			IF iRecValveMode <> 63 AND xDownloadDone = FALSE THEN	// The transfer mode is currently not active and the values are not downloaded yet
				// check whether the WebConfig blocks the access to transfer mode
				fbReadBitsFromWord(wData := awBusDataFromVTEM[0], iStartBit := 8, iEndBit := 15, iValue => iAppStatus);
				IF iRecValveMode = 61 AND iAppStatus = 10 THEN 		// access denied by WebConfig
					xDownloadError := TRUE;
					iResponse := eTransferResponse.access_denied_WebConfig;
					iCommandNumber := 3; 			// do nothing (here: command 'stop')
				ELSIF iRecValveMode = 61 AND iAppStatus = 11 THEN 	// access denied due to an active saving process
					xDownloadError := TRUE;
					iResponse := eTransferResponse.access_denied_saving;
					iCommandNumber := 3; 			// do nothing (here: command 'stop')
				ELSIF iRecValveMode = 61 AND iAppStatus = 15 THEN 	// no valve detected
					xDownloadError := TRUE;
					iResponse := eTransferResponse.no_valve_detected; 
					iCommandNumber := 1; 			// keep downloading (here: command 'download') In a Firmware older than 4.16(E) an empty valve keep sending ValveMode 61 and AppStatus 15. In Firmware 4.16(E) the message changes with a tranfer
				ELSIF iRecValveMode = 61 AND iAppStatus = 0 AND xTransferComplete = TRUE THEN
					// All values are downloaded and the transfer mode has been closed properly
					xDownloadDone := TRUE;
					xDownloadError := FALSE;
					iCommandNumber := 3; 			// command 'stop' to remain the valve stopped
				ELSE	// ready to start transfer mode
					xDownloadError := FALSE;
					iResponse := eTransferResponse.transferring;
					iCommandNumber := 1; 			// command 'download' for the current value
				END_IF
		
			ELSIF iRecValveMode = 63 AND xDownloadDone = FALSE THEN		// The transfer mode is active, but the values are not downloaded yet
				fbReadBitsFromWord(wData := awBusDataFromVTEM[0], iStartBit := 8, iEndBit := 12, iValue => iRecChannel);
				fbReadBitsFromWord(wData := awBusDataFromVTEM[0], iStartBit := 13, iEndBit := 15, iValue => iRecTransferCtrl);
				fbReadBitsFromWord(wData := awBusDataFromVTEM[1], iStartBit := 0, iEndBit := 7, iValue => iRecAddressedTargetType);
				fbReadBitsFromWord(wData := awBusDataFromVTEM[1], iStartBit := 8, iEndBit := 15, iValue => iRecIndex);
				iRecTransferValue := WORD_TO_INT(awBusDataFromVTEM[2]);
		 
				IF aTransferPackages[iCurrentValue].iChannel = iRecChannel AND iRecTransferCtrl = 1 AND aTransferPackages[iCurrentValue].iAddressedTarget = iRecAddressedTargetType AND
					aTransferPackages[iCurrentValue].iIndex = iRecIndex AND  aTransferPackages[iCurrentValue].iTransferValue = iRecTransferValue THEN
						// The download command for the parameter was mirrored by the Motion Terminal, the download has been confirmed
						
						xDownloadError := FALSE;
						iCurrentValue := iCurrentValue +1;		// next value
						
						// check whether there is another value
						IF aTransferPackages[iCurrentValue].iAddressedTarget = 0 AND aTransferPackages[iCurrentValue].iChannel = 0 AND aTransferPackages[iCurrentValue].iIndex = 0 AND
							aTransferPackages[iCurrentValue].iTransferValue = 0 THEN 	// last value reached
							
							iCommandNumber := 2; 		// exit transfer mode
							iResponse := eTransferResponse.transfer_successful;
							xTransferComplete := TRUE;
							xStopPending := TRUE;
						ELSE
							iCommandNumber := 1; 		// command 'download' for the (next) value
							iResponse := eTransferResponse.transferring;
						END_IF
					
				ELSIF iRecChannel = 0 AND iRecTransferCtrl = 0 AND iRecAddressedTargetType = 0 AND iRecIndex = 0 AND iRecTransferValue <> 0 AND xFirstCycle = FALSE THEN
					// An invalid command was sent when using the transfer mode
					
					iCommandNumber := 1; 			// command 'download' for the current value
					xDownloadError := TRUE; 
					
					CASE iRecTransferValue OF		// indicates the type of the invalid command
						1: 	iResponse := eTransferResponse.invalid_Channel;
						2: 	iResponse := eTransferResponse.invalid_TransferControl;	// this should never happen
						3: 	iResponse := eTransferResponse.invalid_AddressedTarget;
						4: 	iResponse := eTransferResponse.invalid_Index;
						5: 	iResponse := eTransferResponse.invalid_TransferValue;
						6: 	iResponse := eTransferResponse.invalid_combination;
						7:  iResponse := eTransferResponse.access_denied_DataInUse;
						8:	iResponse := eTransferResponse.no_data_empty_slot;
					END_CASE
					
				ELSE	// A different value is treated in transfer mode or the command was mirrored wrong
					// waiting for stop ack
					IF xStopPending = FALSE THEN
						iCommandNumber := 1; 			// command 'download' for the current value
						xDownloadError := FALSE;
						iResponse := eTransferResponse.transferring;
					END_IF
				END_IF
			
			ELSE // xDownloadDone = TRUE
				IF aTransferPackages[iCurrentValue].iChannel = 0 AND aTransferPackages[iCurrentValue].iAddressedTarget = 0 AND  aTransferPackages[iCurrentValue].iIndex = 0 AND  aTransferPackages[iCurrentValue].iTransferValue = 0 THEN
					// The FB is still active although all values are already downloaded
					iResponse := eTransferResponse.transfer_successful;
					xDownloadError := FALSE;
					iCommandNumber := 3; 		// do nothing (here: command 'stop', MAs remain stopped)
				ELSE
					// Another set of values was inserted to the FB without resetting the internal state with a falling edge at xExecute before
					iResponse := eTransferResponse.FB_needs_rising_edge_xExecute;
					xDownloadError := TRUE;
					iCommandNumber := 2; 		// do nothing (here: command 'exit transfer mode')
				END_IF
			END_IF
		END_IF
		
	ELSE // xInputValid = FALSE OR xInputConsistent = FALSE
		xDownloadDone := FALSE;
		xDownloadError := TRUE;
		IF iRecValveMode = 63 THEN
			iCommandNumber := 2; 				// command 'exit transfer mode'
		ELSE
			iCommandNumber := 3;				// command 'stop'
		END_IF
	END_IF
	
	xFirstCycle := FALSE;

ELSIF xExecute = FALSE AND xFirstCycle = FALSE THEN			// falling edge at input xExecute, resetting the function block
	IF iRecValveMode = 63 THEN
		iCommandNumber := 2;								// exit transfer mode
	ELSE
		xFirstCycle := TRUE;
		xDownloadDone := FALSE;
		xDownloadError := FALSE;
		xTransferComplete := FALSE;
		iCurrentValue := 0;
		xStopPending := FALSE;
		iResponse := eTransferResponse.ready_for_new_transfer;
		iCommandNumber := 0; 								// do nothing (idle)
	END_IF
		
ELSIF xExecute = FALSE AND xFirstCycle = TRUE THEN			// idle mode for the function block
	iResponse := eTransferResponse.ready_for_new_transfer;
	iCommandNumber := 0;
END_IF

CASE iCommandNumber OF
	0: // idle

	1: // download the current value, addressed and specified in the array of values
		fbWriteValueToWord(iValue := 63, iStartBit := 0, iEndBit := 5, wDataWord := awBusDataToVTEM[0]); 												// ValveMode = 63
		fbWriteValueToWord(iValue := 0, iStartBit := 6, iEndBit := 7, wDataWord := awBusDataToVTEM[0]); 												// (empty)
		fbWriteValueToWord(iValue := aTransferPackages[iCurrentValue].iChannel, iStartBit := 8, iEndBit := 12, wDataWord := awBusDataToVTEM[0]); 		// Channel
		fbWriteValueToWord(iValue := 1, iStartBit := 13, iEndBit := 15, wDataWord := awBusDataToVTEM[0]); 												// TransferControl = download
		fbWriteValueToWord(iValue := aTransferPackages[iCurrentValue].iAddressedTarget, iStartBit := 0, iEndBit := 7, wDataWord := awBusDataToVTEM[1]); 	// AddressedTarget
		fbWriteValueToWord(iValue := aTransferPackages[iCurrentValue].iIndex, iStartBit := 8, iEndBit := 15, wDataWord := awBusDataToVTEM[1]); 			// Index
		
		awBusDataToVTEM[2] := INT_TO_WORD(aTransferPackages[iCurrentValue].iTransferValue);
	
	2: // exit transfer mode
		fbWriteValueToWord(iValue := 63, iStartBit := 0, iEndBit := 5, wDataWord := awBusDataToVTEM[0]); 												// ValveMode = 63
		fbWriteValueToWord(iValue := 0, iStartBit := 6, iEndBit := 7, wDataWord := awBusDataToVTEM[0]); 												// (empty)
		fbWriteValueToWord(iValue := aTransferPackages[iCurrentValue].iChannel, iStartBit := 8, iEndBit := 12, wDataWord := awBusDataToVTEM[0]); 		// Channel
		fbWriteValueToWord(iValue := 3, iStartBit := 13, iEndBit := 15, wDataWord := awBusDataToVTEM[0]); 												// TransferControl = exit

		awBusDataToVTEM[1] := 0; 
		awBusDataToVTEM[2] := 0; 

	3: // stop all Motion Apps
		fbWriteValueToWord(iValue := 61, iStartBit := 0, iEndBit := 5, wDataWord := awBusDataToVTEM[0]); 												// ValveMode = 61
		fbWriteValueToWord(iValue := 0, iStartBit := 6, iEndBit := 15, wDataWord := awBusDataToVTEM[0]); 												// (empty)

		awBusDataToVTEM[1] := 0; 
		awBusDataToVTEM[2] := 0; 
END_CASE

END_FUNCTION_BLOCK

// Transfermode/specific_MA_config/FB_Write_config_MA_04
/// This function block can be used to download the configuration of Motion App 4 ("Model-based proportional pressure regulation").
/// The specific parameters of this Motion App are the inputs of this FB and can be defined by the user. 
/// The function block uses the transfer mode to write this configuration to the Motion Terminal
/// and indicates the state of the download process.

FUNCTION_BLOCK FB_Write_config_MA_04
VAR_INPUT
	awBusDataFromVTEM 				: ARRAY [0..2] OF WORD;		(* 6 bytes of process data received from the Motion Terminal *)
END_VAR

VAR_IN_OUT
	awBusDataToVTEM 				: ARRAY [0..2] OF WORD; 	(* 6 bytes of process data sent to the Motion Terminal *)	
END_VAR

VAR_INPUT
	xExecute 						: BOOL; 					(* has to be set to TRUE for a download and to FALSE to reset the function block after a download *)
		                    		
	iParameterSet					: INT := 1; 				(* the parameter set to be written to, 1 by default *)
	
	// system parameters
		iTubingLengthAt2 			: INT; 						(* length of the tubing connected to outlet port 2 of the valve [1 digit = 1 mm] *)
		iTubingLengthAt4 			: INT;						(* length of the tubing connected to outlet port 4 of the valve [1 digit = 1 mm] *)
		iTubingInnerDiameterAt2 	: INT;  					(* inner diameter of the tubing connected to outlet port 2 of the valve [1 digit = 0.01 mm] *)
		iTubingInnerDiameterAt4 	: INT;						(* inner diameter of the tubing connected to outlet port 4 of the valve [1 digit = 0.01 mm] *)
		iVolumeAt2 					: INT; 						(* size/capacity of the volume connected to outlet port 2 of the valve [1 digit = 0.001 l] *)
	 	iVolumeAt4 					: INT;						(* size/capacity of the volume connected to outlet port 4 of the valve [1 digit = 0.001 l] *)
		iInPortRetracted_optional	: INT;						// Sensor port for detection of end position at pressurisation of outlet port 2 (retracted), value is number of the slot (beginning from 0 and including valve slots) * 10 + number of the port
		iInPortAdvanced_optional	: INT;						// Sensor port for detection of end position at pressurisation of outlet port 4 (advanced), value is number of the slot (beginning from 0 and including valve slots) * 10 + number of the port
    
	// application parameters
		iPressureRiseAt2 			: INT; 						(* maximum pressure rise at outlet port 2 [1 digit = 0.01 bar/s] *)
		iPressureRiseAt4 			: INT;						(* maximum pressure rise at outlet port 4 [1 digit = 0.01 bar/s] *)
END_VAR

VAR_OUTPUT
	iResponse 						: eTransferResponse; 		(* returns the status of the execution of the download process *)
	sCurrentValue 					: STRING; 					(* indicates which value of the array is currently treated (necessary to evaluate in case of error messages) *)
	xDownloadDone 					: BOOL; 					(* indicates whether the download was successful *)
	xDownloadError 					: BOOL := FALSE; 			(* indicates whether an error occurred during the transfer *)
END_VAR

VAR
	aTransferPackages				: ARRAY [0..100] OF stTransferPackage;
	fbdownloadMultipleParameters 	: FB_Download_Multiple_Parameters;
	iCurrentValue					: INT;
	fbWriteValueToWord 				: FB_Write_Value_To_Word;
END_VAR

(*****************************************************************************************************

Festo SE & Co. KG, Esslingen
Copyright (c) 2018. All rights reserved.

Product:            Motion Terminal VTEM
Description:        Function block to download the parameters for Motion App 4 to the Motion Terminal

Object version:     2.00
Last change:        2019-03
======================================================================================================
                                       H I S T O R Y
======================================================================================================
Version:            2.00
Date:               2019-03
Change/Activity:    - added parameters for the sensor port mapping (#2256294)
                    - changed awBusDataToVTEM into VAR_IN_OUT (#2368965)
Release:            3.5.7.230 (CODESYS 3.5.7.2, Lib version 3.0)
Author:             JEBU
------------------------------------------------------------------------------------------------------
Version:            1.00
Date:               2017
Change/Activity:    - created
Release:            3.5.7.220
Author:             HLBG
======================================================================================================

*****************************************************************************************************)

// write the Motion App specific parameters into the struct
	//iTubingLengthAt2
		aTransferPackages[0].iChannel := iParameterSet;
		aTransferPackages[0].iAddressedTarget := 4;
		aTransferPackages[0].iIndex := 12;
		aTransferPackages[0].iTransferValue := iTubingLengthAt2;
	
	//iTubingLengthAt4
		aTransferPackages[1].iChannel := iParameterSet;
		aTransferPackages[1].iAddressedTarget := 4;
		aTransferPackages[1].iIndex := 13;
		aTransferPackages[1].iTransferValue := iTubingLengthAt4;
	
	//iTubingInnerDiameterAt2
		aTransferPackages[2].iChannel := iParameterSet;
		aTransferPackages[2].iAddressedTarget := 4;
		aTransferPackages[2].iIndex := 14;
		aTransferPackages[2].iTransferValue := iTubingInnerDiameterAt2;
	
	//iTubingInnerDiameterAt4
		aTransferPackages[3].iChannel := iParameterSet;
		aTransferPackages[3].iAddressedTarget := 4;
		aTransferPackages[3].iIndex := 15;
		aTransferPackages[3].iTransferValue := iTubingInnerDiameterAt4;
	
	//iVolumeAt2
		aTransferPackages[4].iChannel := iParameterSet;
		aTransferPackages[4].iAddressedTarget := 4;
		aTransferPackages[4].iIndex := 40;
		aTransferPackages[4].iTransferValue := iVolumeAt2;
	
	//iVolumeAt4
		aTransferPackages[5].iChannel := iParameterSet;
		aTransferPackages[5].iAddressedTarget := 4;
		aTransferPackages[5].iIndex := 41;
		aTransferPackages[5].iTransferValue := iVolumeAt4;
	
	//iPressureRiseAt2
		aTransferPackages[6].iChannel := iParameterSet;
		aTransferPackages[6].iAddressedTarget := 4;
		aTransferPackages[6].iIndex := 182;
		aTransferPackages[6].iTransferValue := iPressureRiseAt2;
	
	//iPressureRiseAt4
		aTransferPackages[7].iChannel := iParameterSet;
		aTransferPackages[7].iAddressedTarget := 4;
		aTransferPackages[7].iIndex := 183;
		aTransferPackages[7].iTransferValue := iPressureRiseAt4;
	
	//iInPortRetract_optional
		aTransferPackages[8].iChannel := iParameterSet;
		aTransferPackages[8].iAddressedTarget := 4;
		aTransferPackages[8].iIndex := 70;
		aTransferPackages[8].iTransferValue := iInPortRetracted_optional;
	
	//iInPortAdvanced_optional
		aTransferPackages[9].iChannel := iParameterSet;
		aTransferPackages[9].iAddressedTarget := 4;
		aTransferPackages[9].iIndex := 71;
		aTransferPackages[9].iTransferValue := iInPortAdvanced_optional;
	
	// define end of parameter list to be downloaded by setting all variables to 0 (end criterion for FB_Download_Multiple_Parameters)
		aTransferPackages[10].iChannel := 0;
		aTransferPackages[10].iAddressedTarget := 0;
		aTransferPackages[10].iIndex := 0;
		aTransferPackages[10].iTransferValue := 0;


// pre-check of the value for the parameter set
	IF xExecute = TRUE AND (iParameterSet < 1 OR iParameterSet > 5) THEN		// invalid input for the parameter set
		xDownloadDone := FALSE; 
		xDownloadError := TRUE; 
		iResponse := eTransferResponse.invalid_ParameterSet; 
		iCurrentValue := 0; 
		// send command 'stop'
		fbWriteValueToWord(iValue := 61, iStartBit := 0, iEndBit := 5, wDataWord := awBusDataToVTEM[0]); 			// ValveMode = 61
		fbWriteValueToWord(iValue := 0, iStartBit := 6, iEndBit := 15, wDataWord := awBusDataToVTEM[0]); 			// (empty)
		awBusDataToVTEM[1] := 0; 
		awBusDataToVTEM[2] := 0; 
		
	ELSE	
		// call the function block for multiple parameter download
			fbdownloadMultipleParameters(	xExecute := xExecute,
											awBusDataFromVTEM := awBusDataFromVTEM,
											aTransferPackages := aTransferPackages, 
											awBusDataToVTEM := awBusDataToVTEM,
											xDownloadDone => xDownloadDone,
											xDownloadError => xDownloadError,
											iResponse => iResponse,
											iCurrentValue => iCurrentValue);
	END_IF
	

// The current value output is needed if there is any invalid value in order to address it correctly.
// As the user doesn't work with indices in this function block, the current value is transformed to a string holding the name of the parameter.
	CASE iCurrentValue OF
		0: sCurrentValue := 'iTubingLengthAt2';
		1: sCurrentValue := 'iTubingLengthAt4';
		2: sCurrentValue := 'iTubingInnerDiameterAt2';
		3: sCurrentValue := 'iTubingInnerDiameterAt4';
		4: sCurrentValue := 'iVolumeAt2';
		5: sCurrentValue := 'iVolumeAt4';
		6: sCurrentValue := 'iPressureRiseAt2';
		7: sCurrentValue := 'iPressureRiseAt4';
		8: sCurrentValue := 'iInPortRetract_optional';
		9: sCurrentValue := 'iInPortAdvanced_optional';
		10: sCurrentValue := 'AllParametersWritten';
	END_CASE

END_FUNCTION_BLOCK

// Transfermode/specific_MA_config/FB_Write_config_MA_11
/// This function block can be used to download the configuration of Motion App 11 ("Soft stop").
/// The specific parameters of this Motion App are the inputs of this FB and can be defined by the user. 
/// The function block uses the transfer mode to write this configuration to the Motion Terminal
/// and indicates the state of the download process.

FUNCTION_BLOCK FB_Write_config_MA_11
VAR_INPUT
	awBusDataFromVTEM 				: ARRAY [0..2] OF WORD;		(* 6 bytes of process data received from the Motion Terminal *)
END_VAR

VAR_IN_OUT
	awBusDataToVTEM					: ARRAY [0..2] OF WORD; 	(* 6 bytes of process data sent to the Motion Terminal *)
END_VAR

VAR_INPUT
	xExecute 						: BOOL; 					(* has to be set to TRUE for a download and to FALSE to reset the function block after a download *)
	
	iParameterSet					: INT := 1; 				(* the parameter set to be written to, 1 by default *)
	
	// system parameters
		iDriveType 					: INT;						// type of the drive/cylinder/... that is to be operated by the valve ->  see list of drive types at support portal (www.festo.com/sp/)
	 	iDriveStroke 				: INT; 						(* stroke of the drive/cylinder/... that is to be operated by the valve [1 digit = 1 mm for linear drives, 1 digit = 1° for rotary drives] *)
		iInstallationPositionDrive 	: INT;  	 				(* inclination of the cylinder with reference to a horizontal installation position [1 digit = 0.01°, positive values = advancing upwards] *)
		iInPortRetracted			: INT;						// Sensor port for detection of end position at pressurisation of outlet port 2 (retracted), value is number of the slot (beginning from 0 and including valve slots) * 10 + number of the port
		iInPortAdvanced				: INT;						// Sensor port for detection of end position at pressurisation of outlet port 4 (advanced), value is number of the slot (beginning from 0 and including valve slots) * 10 + number of the port
	
	// application parameters                               	
	 	iLoadAdvancing 				: INT := 0; 				(* mass that is to be moved by the drive when advancing ((4) pressurised) [1 digit = 0.01 kg] *)
		iLoadRetracting 			: INT := 0;					(* mass that is to be moved by the drive when retracting ((2) pressurised) [1 digit = 0.01 kg] *)

END_VAR

VAR_OUTPUT                                                  	
	iResponse 						: eTransferResponse; 		(* returns the status of the execution of the download process *)
	sCurrentValue 					: STRING; 					(* indicates which value of the array is currently treated (necessary to evaluate in case of error messages) *)
	xDownloadDone 					: BOOL; 					(* indicates whether the download was successful *)
	xDownloadError 					: BOOL := FALSE; 			(* indicates whether an error occurred during the transfer *)
END_VAR

VAR
	aTransferPackages				: ARRAY [0..100] OF stTransferPackage;
	fbdownloadMultipleParameters 	: FB_Download_Multiple_Parameters;
	iCurrentValue					: INT;
	fbWriteValueToWord 				: FB_Write_Value_To_Word;
END_VAR

(*****************************************************************************************************

Festo SE & Co. KG, Esslingen
Copyright (c) 2018. All rights reserved.

Product:            Motion Terminal VTEM
Description:        Function block to download the parameters for Motion App 11 to the Motion Terminal

Object version:     2.01
Last change:        2019-03
======================================================================================================
                                       H I S T O R Y
======================================================================================================
Version:            2.01
Date:               2019-03
Change/Activity:    - sensor port mapping parameters (#2397241)
Release:            3.5.7.231 (CODESYS 3.5.7.2, Lib version 3.1)
Author:             JEBU
------------------------------------------------------------------------------------------------------
Version:            2.00
Date:               2019-03
Change/Activity:    - added parameters for the sensor port mapping (#2256294)
                    - removed tuning parameters (#2374189)
                    - changed awBusDataToVTEM into VAR_IN_OUT (#2368965)
Release:            3.5.7.230 (CODESYS 3.5.7.2, Lib version 3.0)
Author:             JEBU
------------------------------------------------------------------------------------------------------
Version:            1.01
Date:               2018-08
Change/Activity:    - added tuning parameters
Release:            3.5.7.220
Author:             JEBU
------------------------------------------------------------------------------------------------------
Version:            1.00
Date:               2017
Change/Activity:    - created
Release:            not released
Author:             HLBG
======================================================================================================

*****************************************************************************************************)

// write the Motion App specific parameters into the struct
	//iDriveType
		aTransferPackages[0].iChannel := iParameterSet;
		aTransferPackages[0].iAddressedTarget := 11;
		aTransferPackages[0].iIndex := 20;
		aTransferPackages[0].iTransferValue := iDriveType;
		
	//iDriveStroke
		aTransferPackages[1].iChannel := iParameterSet;
		aTransferPackages[1].iAddressedTarget := 11;
		aTransferPackages[1].iIndex := 21;
		aTransferPackages[1].iTransferValue := iDriveStroke;
		
	//iInstallationPositionDrive
		aTransferPackages[2].iChannel := iParameterSet;
		aTransferPackages[2].iAddressedTarget := 11;
		aTransferPackages[2].iIndex := 60;
		aTransferPackages[2].iTransferValue := iInstallationPositionDrive;
		
	//iLoadAdvancing
		aTransferPackages[3].iChannel := iParameterSet;
		aTransferPackages[3].iAddressedTarget := 11;
		aTransferPackages[3].iIndex := 101;
		aTransferPackages[3].iTransferValue := iLoadAdvancing;
		
	//iLoadRetracting
		aTransferPackages[4].iChannel := iParameterSet;
		aTransferPackages[4].iAddressedTarget := 11;
		aTransferPackages[4].iIndex := 100;
		aTransferPackages[4].iTransferValue := iLoadRetracting;
		
	//iInPortRetract
		aTransferPackages[5].iChannel := iParameterSet;
		aTransferPackages[5].iAddressedTarget := 11;
		aTransferPackages[5].iIndex := 75;
		aTransferPackages[5].iTransferValue := iInPortRetracted;
	
	//iInPortRetract
		aTransferPackages[6].iChannel := iParameterSet;
		aTransferPackages[6].iAddressedTarget := 11;
		aTransferPackages[6].iIndex := 76;
		aTransferPackages[6].iTransferValue := iInPortAdvanced;
	
	// define end of parameter list to be downloaded by setting all variables to 0 (end criterion for FB_Download_Multiple_Parameters)
		aTransferPackages[7].iChannel := 0;
		aTransferPackages[7].iAddressedTarget := 0;
		aTransferPackages[7].iIndex := 0;
		aTransferPackages[7].iTransferValue := 0;


// pre-check of the value for the parameter set
	IF xExecute = TRUE AND (iParameterSet < 1 OR iParameterSet > 5) THEN		// invalid input for the parameter set
		xDownloadDone := FALSE; 
		xDownloadError := TRUE; 
		iResponse := eTransferResponse.invalid_ParameterSet; 
		iCurrentValue := 0; 
		// send command 'stop'
		fbWriteValueToWord(iValue := 61, iStartBit := 0, iEndBit := 5, wDataWord := awBusDataToVTEM[0]); 			// ValveMode = 61
		fbWriteValueToWord(iValue := 0, iStartBit := 6, iEndBit := 15, wDataWord := awBusDataToVTEM[0]); 			// (empty)
		awBusDataToVTEM[1] := 0; 
		awBusDataToVTEM[2] := 0; 
		
	ELSE	
		// call the function block for multiple parameter download
			fbdownloadMultipleParameters(	xExecute := xExecute,
											awBusDataFromVTEM := awBusDataFromVTEM,
											aTransferPackages := aTransferPackages, 
											awBusDataToVTEM := awBusDataToVTEM,
											xDownloadDone => xDownloadDone,
											xDownloadError => xDownloadError,
											iResponse => iResponse,
											iCurrentValue => iCurrentValue);
	END_IF
		
	
// The current value output is needed if there is any invalid value in order to address it correctly.
// As the user doesn't work with indices in this function block, the current value is transformed to a string holding the name of the parameter.
	CASE iCurrentValue OF
		0: sCurrentValue := 'iDriveType';
		1: sCurrentValue := 'iDriveStroke';
		2: sCurrentValue := 'iInstallationPositionDrive';
		3: sCurrentValue := 'iLoadAdvancing';
		4: sCurrentValue := 'iLoadRetracting';
		5: sCurrentValue := 'iInPortRetract';
		6: sCurrentValue := 'iInPortAdvanced';
		7: sCurrentValue := 'AllParametersWritten';
	END_CASE

END_FUNCTION_BLOCK

// Transfermode/specific_MA_config/FB_Write_config_MA_12
/// This function block can be used to download the configuration of Motion App 12 ("Leakage diagnostics").
/// The specific parameters of this Motion App are the inputs of this FB and can be defined by the user. 
/// The function block uses the transfer mode to write this configuration to the Motion Terminal
/// and indicates the state of the download process.

FUNCTION_BLOCK FB_Write_config_MA_12
VAR_INPUT
	awBusDataFromVTEM 				: ARRAY [0..2] OF WORD;		(* 6 bytes of process data received from the Motion Terminal *)
END_VAR

VAR_IN_OUT
	awBusDataToVTEM 				: ARRAY [0..2] OF WORD; 	(* 6 bytes of process data sent to the Motion Terminal *)
END_VAR

VAR_INPUT
	xExecute 						: BOOL; 					(* has to be set to TRUE for a download and to FALSE to reset the function block after a download *)
		                                                    	
	iParameterSet					: INT := 1; 				(* the parameter set to be written to, 1 by default *)
	
	// system parameters
		iTubingLengthAt2 			: INT; 						(* length of the tubing connected to outlet port 2 of the valve [1 digit = 1 mm] *)
	 	iTubingLengthAt4 			: INT;						(* length of the tubing connected to outlet port 4 of the valve [1 digit = 1 mm] *)
	 	iTubingInnerDiameterAt2		: INT;  					(* inner diameter of the tubing connected to outlet port 2 of the valve [1 digit = 0.01mm] *)
	 	iTubingInnerDiameterAt4		: INT;						(* inner diameter of the tubing connected to outlet port 4 of the valve [1 digit = 0.01mm] *)
	 	iDriveType 					: INT;						// type of the drive/cylinder/... that is to be operated by the valve ->  see list of drive types at support portal (www.festo.com/sp/)
	 	iDriveStroke 				: INT; 						(* stroke of the drive/cylinder/... that is to be operated by the valve [1 digit = 1 mm for linear drives, 1 digit = 1° for rotary drives] *)
		iVolumeAt2 					: INT; 						(* size/capacity of the volume connected to outlet port 2 of the valve [1 digit = 0.001 l] *)
		iVolumeAt4 					: INT;						(* size/capacity of the volume connected to outlet port 4 of the valve [1 digit = 0.001 l] *)
		iInstallationPositionDrive 	: INT;  	 				(* inclination of the cylinder with reference to a horizontal installation position [1 digit = 0.01°, positive values = advancing upwards] *)

	// application parameters                               	
		iLoadRetracting 			: INT;						(* mass that is to be moved by the drive when retracting ((2) pressurised) [1 digit = 0.01 kg] *)
	 	iLoadAdvancing 				: INT; 						(* mass that is to be moved by the drive when advancing ((4) pressurised) [1 digit = 0.01 kg] *)
		iMomentOfInertiaRetracting	: INT;						// Moment of inertia during for swivel drives when retratcting ((2) pressirised) [1 digit = 1 kg cm³]
		iMomentOfInertiaAdvancing	: INT;						// Moment of inertia during for swivel drives when advancing ((4) pressirised) [1 digit = 1 kg cm³]
		iMaxLeakageForStatusGood 	: INT;						(* allowed deviation regarding reference value for status "Good" [1 digit = 0.1 l/h] *)
		iMaxLeakageForStatusWarning : INT;						(* allowed deviation regarding reference value for status "Warning" [1 digit = 0.1 l/h] *)
	 	iMaxLeakageForStatusCritical: INT; 						(* allowed deviation regarding reference value for status "Critical" [1 digit = 0.1 l/h] *)
END_VAR

VAR_OUTPUT                                                  	
	iResponse 						: eTransferResponse;		(* returns the status of the execution of the download process *)
	sCurrentValue 					: STRING; 					(* indicates which value of the array is currently treated (necessary to evaluate in case of error messages) *)
	xDownloadDone 					: BOOL; 					(* indicates whether the download was successful *)
	xDownloadError 					: BOOL := FALSE; 			(* indicates whether an error occurred during the transfer *)
END_VAR

VAR
	aTransferPackages				: ARRAY [0..100] OF stTransferPackage;
	fbdownloadMultipleParameters 	: FB_Download_Multiple_Parameters;
	iCurrentValue					: INT;
	fbWriteValueToWord 				: FB_Write_Value_To_Word;
END_VAR

(*****************************************************************************************************

Festo SE & Co. KG, Esslingen
Copyright (c) 2018. All rights reserved.

Product:            Motion Terminal VTEM
Description:        Function block to download the parameters for Motion App 12 to the Motion Terminal

Object version:     2.01
Last change:        2019-04
======================================================================================================
                                       H I S T O R Y
======================================================================================================
Version:            2.01
Date:               2019-04
Change/Activity:    - added parameters for moment of inertia used for swivel drives (#2307852)
                    - changed awBusDataToVTEM into VAR_IN_OUT (#2368965)
Release:            3.5.7.231 (CODESYS 3.5.7.2, Lib version 3.1)
Author:             JEBU
------------------------------------------------------------------------------------------------------
Version:            1.00
Date:               2017
Change/Activity:    - created
Release:            3.5.7.22 (CODESYS 3.5.7.2, Lib version 2.0)
Author:             HLBG
======================================================================================================

*****************************************************************************************************)

// write the Motion App specific parameters into the struct
	//iTubingLengthAt2
		aTransferPackages[0].iChannel := iParameterSet;
		aTransferPackages[0].iAddressedTarget := 12;
		aTransferPackages[0].iIndex := 12;
		aTransferPackages[0].iTransferValue := iTubingLengthAt2;
		
	//iTubingLengthAt4
		aTransferPackages[1].iChannel := iParameterSet;
		aTransferPackages[1].iAddressedTarget := 12;
		aTransferPackages[1].iIndex := 13;
		aTransferPackages[1].iTransferValue := iTubingLengthAt4;
		
	//iTubingInnerDiameterAt2
		aTransferPackages[2].iChannel := iParameterSet;
		aTransferPackages[2].iAddressedTarget := 12;
		aTransferPackages[2].iIndex := 14;
		aTransferPackages[2].iTransferValue := iTubingInnerDiameterAt2;
		
	//iTubingInnerDiameterAt4
		aTransferPackages[3].iChannel := iParameterSet;
		aTransferPackages[3].iAddressedTarget := 12;
		aTransferPackages[3].iIndex := 15;
		aTransferPackages[3].iTransferValue := iTubingInnerDiameterAt4;
		
	//iDriveType
		aTransferPackages[4].iChannel := iParameterSet;
		aTransferPackages[4].iAddressedTarget := 12;
		aTransferPackages[4].iIndex := 20;
		aTransferPackages[4].iTransferValue := iDriveType;
		
	//iDriveStroke
		aTransferPackages[5].iChannel := iParameterSet;
		aTransferPackages[5].iAddressedTarget := 12;
		aTransferPackages[5].iIndex := 21;
		aTransferPackages[5].iTransferValue := iDriveStroke;
		
	//iVolumeAt2
		aTransferPackages[6].iChannel := iParameterSet;
		aTransferPackages[6].iAddressedTarget := 12;
		aTransferPackages[6].iIndex := 40;
		aTransferPackages[6].iTransferValue := iVolumeAt2;
		
	//iVolumeAt4 
		aTransferPackages[7].iChannel := iParameterSet;
		aTransferPackages[7].iAddressedTarget := 12;
		aTransferPackages[7].iIndex := 41;
		aTransferPackages[7].iTransferValue := iVolumeAt4;
		
	//iInstallationPositionDrive
		aTransferPackages[8].iChannel := iParameterSet;
		aTransferPackages[8].iAddressedTarget := 12;
		aTransferPackages[8].iIndex := 60;
		aTransferPackages[8].iTransferValue := iInstallationPositionDrive;
		
	//iLoadRetracting
		aTransferPackages[9].iChannel := iParameterSet;
		aTransferPackages[9].iAddressedTarget := 12;
		aTransferPackages[9].iIndex := 100;
		aTransferPackages[9].iTransferValue := iLoadRetracting;
		
	//iLoadAdvancing
		aTransferPackages[10].iChannel := iParameterSet;
		aTransferPackages[10].iAddressedTarget := 12;
		aTransferPackages[10].iIndex := 101;
		aTransferPackages[10].iTransferValue := iLoadAdvancing;
		
	//iMomentOfInertiaRetracting
		aTransferPackages[11].iChannel := iParameterSet;
		aTransferPackages[11].iAddressedTarget := 12;
		aTransferPackages[11].iIndex := 102;
		aTransferPackages[11].iTransferValue := iMomentOfInertiaRetracting;
	
	//iMomentOfInertiaAdvancing
		aTransferPackages[12].iChannel := iParameterSet;
		aTransferPackages[12].iAddressedTarget := 12;
		aTransferPackages[12].iIndex := 103;
		aTransferPackages[12].iTransferValue := iMomentOfInertiaAdvancing;

	//iMaxLeakageForStatusGood
		aTransferPackages[13].iChannel := iParameterSet;
		aTransferPackages[13].iAddressedTarget := 12;
		aTransferPackages[13].iIndex := 200;
		aTransferPackages[13].iTransferValue := iMaxLeakageForStatusGood;
		
	//iMaxLeakageForStatusWarning
		aTransferPackages[14].iChannel := iParameterSet;
		aTransferPackages[14].iAddressedTarget := 12;
		aTransferPackages[14].iIndex := 201;
		aTransferPackages[14].iTransferValue := iMaxLeakageForStatusWarning;
		
	//iMaxLeakageForStatusCritical
		aTransferPackages[15].iChannel := iParameterSet;
		aTransferPackages[15].iAddressedTarget := 12;
		aTransferPackages[15].iIndex := 202;
		aTransferPackages[15].iTransferValue := iMaxLeakageForStatusCritical;
	
	// define end of parameter list to be downloaded by setting all variables to 0 (end criterion for FB_Download_Multiple_Parameters)
		aTransferPackages[16].iChannel := 0;
		aTransferPackages[16].iAddressedTarget := 0;
		aTransferPackages[16].iIndex := 0;
		aTransferPackages[16].iTransferValue := 0;


// pre-check of the value for the parameter set
	IF xExecute = TRUE AND (iParameterSet < 1 OR iParameterSet > 5) THEN		// invalid input for the parameter set
		xDownloadDone := FALSE; 
		xDownloadError := TRUE; 
		iResponse := eTransferResponse.invalid_ParameterSet; 
		iCurrentValue := 0; 
		// send command 'stop'
		fbWriteValueToWord(iValue := 61, iStartBit := 0, iEndBit := 5, wDataWord := awBusDataToVTEM[0]); 			// ValveMode = 61
		fbWriteValueToWord(iValue := 0, iStartBit := 6, iEndBit := 15, wDataWord := awBusDataToVTEM[0]); 			// (empty)
		awBusDataToVTEM[1] := 0; 
		awBusDataToVTEM[2] := 0; 
		
	ELSE	
		// call the function block for multiple parameter download
			fbdownloadMultipleParameters(	xExecute := xExecute,
											awBusDataFromVTEM := awBusDataFromVTEM,
											aTransferPackages := aTransferPackages, 
											awBusDataToVTEM := awBusDataToVTEM,
											xDownloadDone => xDownloadDone,
											xDownloadError => xDownloadError,
											iResponse => iResponse,
											iCurrentValue => iCurrentValue);
	END_IF
		
	
// The current value output is needed if there is any invalid value in order to address it correctly.
// As the user doesn't work with indices in this function block, the current value is transformed to a string holding the name of the parameter.
	CASE iCurrentValue OF
		0: sCurrentValue := 'iTubingLengthAt2';
		1: sCurrentValue := 'iTubingLengthAt4';
		2: sCurrentValue := 'iTubingInnerDiameterAt2';
		3: sCurrentValue := 'iTubingInnerDiameterAt4';
		4: sCurrentValue := 'iDriveType';
		5: sCurrentValue := 'iDriveStroke';
		6: sCurrentValue := 'iVolumeAt2';
		7: sCurrentValue := 'iVolumeAt4';
		8: sCurrentValue := 'iInstallationPositionDrive';
		9: sCurrentValue := 'iLoadRetracting';
		10: sCurrentValue := 'iLoadAdvancing';
		11: sCurrentValue := 'iMomentOfInertiaRetracting';
		12: sCurrentValue := 'iMomentOfInertiaAdvancing';
		13: sCurrentValue := 'iMaxLeakageForStatusGood';
		14: sCurrentValue := 'iMaxLeakageForStatusWarning';
		15: sCurrentValue := 'iMaxLeakageForStatusCritical';
		16: sCurrentValue := 'AllParametersWritten';
	END_CASE

END_FUNCTION_BLOCK

// StateInterpreter/FB_StateInterpreter_MA_02
/// The variable "byActualAppState" is an output of the FB_ValveControl that is used differently in each Motion App.
/// This function block interprets the "AppState" output of the FB_ValveControl if Motion App 2 ("Proportional directional control valve") is running.
/// The Motion App specific values are derived from the "byActualAppState".

FUNCTION_BLOCK FB_StateInterpreter_MA_02
VAR_INPUT
	byActualAppState 			: BYTE; 	(* output of the FB_ValveControl *)
END_VAR
VAR_OUTPUT
	xMeaningOfActVal1			: BOOL;		// Indicates which information about outlet port (2) is output with actual value 1. 0 = valve position [1 digit = 0.01%], 1 = relative pressure [1 digit = 1 mbar]
	xMeaningOfActVal2			: BOOL;		// Indicates which information about outlet port (4) is output with actual value 2. 0 = valve position [1 digit = 0.01%], 1 = relative pressure [1 digit = 1 mbar]
	xRetractedEndPos_optional	: BOOL;  	(* only if digital sensors are installed (optional): indicates whether the retracted end position was reached (after outlet port 2 is pressurised) *)
	xAdvancedEndPos_optional	: BOOL;  	(* only if digital sensors are installed (optional): indicates whether the advanced end position was reached (after outlet port 4 is pressurised) *)
	xWarning					: BOOL; 	(* indicates whether there is a warning returned by the Motion App *)
END_VAR
VAR
	fbReadBitsFromByte			: FB_Read_Bits_From_Byte;
	byMeaningOfActVal1			: BYTE;
	byMeaningOfActVal2	: BYTE;
	byRetractedEndPos			: BYTE;
	byAdvancedEndPos			: BYTE;
	byWarning					: BYTE;
END_VAR

(*****************************************************************************************************

Festo SE & Co. KG, Esslingen
Copyright (c) 2018. All rights reserved.

Product:            Motion Terminal VTEM
Description:        Function block for interpreting the app state of Motion App 2

Object version:     1.01
Last change:        2020-11
======================================================================================================
                                       H I S T O R Y
======================================================================================================
Version:            1.01
Date:               2020-11
Change/Activity:    - added outputs for indicating meaning of actual values (#3797793)
Release:            3.5.7.236
Author:             JEBU
------------------------------------------------------------------------------------------------------
Version:            1.00
Date:               2017
Change/Activity:    - created
Release:            3.5.7.220
Author:             HLBG
======================================================================================================

*****************************************************************************************************)

// read the Motion App specific values from the ActualAppState byte
fbReadBitsFromByte(byData := byActualAppState, iStartBit := 5, iEndBit := 5, byValue => byMeaningOfActVal1);
xMeaningOfActVal1 :=  BYTE_TO_BIT(byMeaningOfActVal1);

fbReadBitsFromByte(byData := byActualAppState, iStartBit := 6, iEndBit := 6, byValue => byMeaningOfActVal2);
xMeaningOfActVal2 :=  BYTE_TO_BIT(byMeaningOfActVal2);

fbReadBitsFromByte(byData := byActualAppState, iStartBit := 0, iEndBit := 0, byValue => byRetractedEndPos);
xRetractedEndPos_optional :=  BYTE_TO_BIT(byRetractedEndPos);

fbReadBitsFromByte(byData := byActualAppState, iStartBit := 2, iEndBit := 2, byValue => byAdvancedEndPos); 
xAdvancedEndPos_optional :=  BYTE_TO_BIT(byAdvancedEndPos);

fbReadBitsFromByte(byData := byActualAppState, iStartBit := 7, iEndBit := 7, byValue => byWarning);
xWarning := BYTE_TO_BIT(byWarning);

END_FUNCTION_BLOCK

// StateInterpreter/FB_StateInterpreter_MA_03
/// The variable "byActualAppState" is an output of the FB_ValveControl that is used differently in each Motion App.
/// This function block interprets the "AppState" output of the FB_ValveControl if Motion App 3 ("Proportional pressure regulation") is running.
/// The Motion App specific values are derived from the "byActualAppState".

FUNCTION_BLOCK FB_StateInterpreter_MA_03
VAR_INPUT
	byActualAppState 			: BYTE; 	(* output of the FB_ValveControl *)
END_VAR
VAR_OUTPUT
	xRetractedEndPos_optional	: BOOL;  	(* only if digital sensors are installed (optional): indicates whether the retracted end position was reached (after outlet port 2 is pressurised) *)
	xAdvancedEndPos_optional	: BOOL;  	(* only if digital sensors are installed (optional): indicates whether the advanced end position was reached (after outlet port 4 is pressurised) *)
	xWarning					: BOOL; 	(* indicates whether there is a warning returned by the Motion App *)
END_VAR
VAR
	fbReadBitsFromByte			: FB_Read_Bits_From_Byte;
	byRetractedEndPos			: BYTE;
	byAdvancedEndPos			: BYTE;
	byWarning					: BYTE;
END_VAR

(*****************************************************************************************************

Festo SE & Co. KG, Esslingen
Copyright (c) 2018. All rights reserved.

Product:            Motion Terminal VTEM
Description:        Function block for interpreting the app state of Motion App 3

Object version:     1.00
Last change:        2017
======================================================================================================
                                       H I S T O R Y
======================================================================================================
Version:            1.00
Date:               2017
Change/Activity:    - created
Release:            3.5.7.220
Author:             HLBG
======================================================================================================

*****************************************************************************************************)

// read the Motion App specific values from the ActualAppState byte
fbReadBitsFromByte(byData := byActualAppState, iStartBit := 0, iEndBit := 0, byValue => byRetractedEndPos);
xRetractedEndPos_optional :=  BYTE_TO_BIT(byRetractedEndPos);

fbReadBitsFromByte(byData := byActualAppState, iStartBit := 2, iEndBit := 2, byValue => byAdvancedEndPos); 
xAdvancedEndPos_optional :=  BYTE_TO_BIT(byAdvancedEndPos);

fbReadBitsFromByte(byData := byActualAppState, iStartBit := 7, iEndBit := 7, byValue => byWarning);
xWarning := BYTE_TO_BIT(byWarning);

END_FUNCTION_BLOCK

// StateInterpreter/FB_StateInterpreter_MA_04
/// The variable "byActualAppState" is an output of the FB_ValveControl that is used differently in each Motion App.
/// This function block interprets the "AppState" output of the FB_ValveControl if Motion App 4 ("Model-based proportional pressure regulation") is running.
/// The Motion App specific values are derived from the "byActualAppState".

FUNCTION_BLOCK FB_StateInterpreter_MA_04
VAR_INPUT
	byActualAppState 			: BYTE; 	(* output of the FB_ValveControl *)
END_VAR
VAR_OUTPUT
	xRetractedEndPos_optional	: BOOL;  	(* only if digital sensors are installed (optional): indicates whether the retracted end position was reached (after outlet port 2 is pressurised) *)
	xAdvancedEndPos_optional	: BOOL;  	(* only if digital sensors are installed (optional): indicates whether the advanced end position was reached (after outlet port 4 is pressurised) *)
	xWarning					: BOOL; 	(* indicates whether there is a warning returned by the Motion App *)
END_VAR
VAR
	fbReadBitsFromByte			: FB_Read_Bits_From_Byte;
	byRetractedEndPos			: BYTE;
	byAdvancedEndPos			: BYTE;
	byWarning					: BYTE;
END_VAR

(*****************************************************************************************************

Festo SE & Co. KG, Esslingen
Copyright (c) 2018. All rights reserved.

Product:            Motion Terminal VTEM
Description:        Function block for interpreting the app state of Motion App 4

Object version:     1.00
Last change:        2017
======================================================================================================
                                       H I S T O R Y
======================================================================================================
Version:            1.00
Date:               2017
Change/Activity:    - created
Release:            3.5.7.220
Author:             HLBG
======================================================================================================

*****************************************************************************************************)

// read the Motion App specific values from the ActualAppState byte
fbReadBitsFromByte(byData := byActualAppState, iStartBit := 0, iEndBit := 0, byValue => byRetractedEndPos);
xRetractedEndPos_optional :=  BYTE_TO_BIT(byRetractedEndPos);

fbReadBitsFromByte(byData := byActualAppState, iStartBit := 2, iEndBit := 2, byValue => byAdvancedEndPos); 
xAdvancedEndPos_optional :=  BYTE_TO_BIT(byAdvancedEndPos);

fbReadBitsFromByte(byData := byActualAppState, iStartBit := 7, iEndBit := 7, byValue => byWarning);
xWarning := BYTE_TO_BIT(byWarning);

END_FUNCTION_BLOCK

// StateInterpreter/FB_StateInterpreter_MA_05
/// The variable "byActualAppState" is an output of the FB_ValveControl that is used differently in each Motion App.
/// This function block interprets the "AppState" output of the FB_ValveControl if Motion App 5 ("Supply and exhaust air flow control") is running.
/// The Motion App specific values are derived from the "byActualAppState".

FUNCTION_BLOCK FB_StateInterpreter_MA_05
VAR_INPUT
	byActualAppState 			: BYTE; 	(* output of the FB_ValveControl *)
END_VAR
VAR_OUTPUT
	xMeaningOfActVal1			: BOOL;		// Indicates which information about outlet port (2) is output with actual value 1. 0 = opening degree exhaust air flow [1 digit = 0.01%], 1 = relative pressure [1 digit = 1 mbar]
	xMeaningOfActVal2			: BOOL;		// Indicates which information about outlet port (4) is output with actual value 2. 0 = opening degree supply air flow [1 digit = 0.01%], 1 = relative pressure [1 digit = 1 mbar]
	xRetractedEndPos_optional	: BOOL;  	(* only if digital sensors are installed (optional): indicates whether the retracted end position was reached (after outlet port 2 is pressurised) *)
	xAdvancedEndPos_optional	: BOOL;  	(* only if digital sensors are installed (optional): indicates whether the advanced end position was reached (after outlet port 4 is pressurised) *)
	xWarning					: BOOL; 	(* indicates whether there is a warning returned by the Motion App *)
END_VAR
VAR
	fbReadBitsFromByte			: FB_Read_Bits_From_Byte;
	byMeaningOfActVal1	: BYTE;
	byMeaningOfActVal2	: BYTE;
	byRetractedEndPos			: BYTE;
	byAdvancedEndPos			: BYTE;
	byWarning					: BYTE;
END_VAR

(*****************************************************************************************************

Festo SE & Co. KG, Esslingen
Copyright (c) 2018. All rights reserved.

Product:            Motion Terminal VTEM
Description:        Function block for interpreting the app state of Motion App 5 

Object version:     1.01
Last change:        2020-11
======================================================================================================
                                       H I S T O R Y
======================================================================================================
Version:            1.01
Date:               2020-11
Change/Activity:    - added outputs for indicating meaning of actual values (#3797793)
Release:            3.5.7.236
Author:             JEBU
------------------------------------------------------------------------------------------------------
Version:            1.00
Date:               2017
Change/Activity:    - created
Release:            3.5.7.220
Author:             HLBG
======================================================================================================

*****************************************************************************************************)

// read the Motion App specific values from the ActualAppState byte
fbReadBitsFromByte(byData := byActualAppState, iStartBit := 5, iEndBit := 5, byValue => byMeaningOfActVal1);
xMeaningOfActVal1 :=  BYTE_TO_BIT(byMeaningOfActVal1);

fbReadBitsFromByte(byData := byActualAppState, iStartBit := 6, iEndBit := 6, byValue => byMeaningOfActVal2);
xMeaningOfActVal2 :=  BYTE_TO_BIT(byMeaningOfActVal2);

fbReadBitsFromByte(byData := byActualAppState, iStartBit := 0, iEndBit := 0, byValue => byRetractedEndPos);
xRetractedEndPos_optional :=  BYTE_TO_BIT(byRetractedEndPos);

fbReadBitsFromByte(byData := byActualAppState, iStartBit := 2, iEndBit := 2, byValue => byAdvancedEndPos); 
xAdvancedEndPos_optional :=  BYTE_TO_BIT(byAdvancedEndPos);

fbReadBitsFromByte(byData := byActualAppState, iStartBit := 7, iEndBit := 7, byValue => byWarning);
xWarning := BYTE_TO_BIT(byWarning);

END_FUNCTION_BLOCK

// StateInterpreter/FB_StateInterpreter_MA_08
/// The variable "byActualAppState" is an output of the FB_ValveControl that is used differently in each Motion App.
/// This function block interprets the "AppState" output of the FB_ValveControl if Motion App 8 ("Selectable pressure level (ECO)") is running.
/// The Motion App specific values are derived from the "byActualAppState".

FUNCTION_BLOCK FB_StateInterpreter_MA_08
VAR_INPUT
	byActualAppState 			: BYTE; 	(* output of the FB_ValveControl *)
END_VAR
VAR_OUTPUT
	xRetractedEndPos_optional	: BOOL;  	(* only if digital sensors are installed (optional): indicates whether the retracted end position was reached (after outlet port 2 is pressurised) *)
	xAdvancedEndPos_optional	: BOOL;  	(* only if digital sensors are installed (optional): indicates whether the advanced end position was reached (after outlet port 4 is pressurised) *)
	xWarning					: BOOL; 	(* indicates whether there is a warning returned by the Motion App *)
END_VAR
VAR
	fbReadBitsFromByte			: FB_Read_Bits_From_Byte;
	byRetractedEndPos			: BYTE;
	byAdvancedEndPos			: BYTE;
	byWarning					: BYTE;
END_VAR

(*****************************************************************************************************

Festo SE & Co. KG, Esslingen
Copyright (c) 2018. All rights reserved.

Product:            Motion Terminal VTEM
Description:        Function block for interpreting the app state of Motion App 8 

Object version:     1.00
Last change:        2017
======================================================================================================
                                       H I S T O R Y
======================================================================================================
Version:            1.00
Date:               2017
Change/Activity:    - created
Release:            3.5.7.220
Author:             HLBG
======================================================================================================

*****************************************************************************************************)

// read the Motion App specific values from the ActualAppState byte
fbReadBitsFromByte(byData := byActualAppState, iStartBit := 0, iEndBit := 0, byValue => byRetractedEndPos);
xRetractedEndPos_optional :=  BYTE_TO_BIT(byRetractedEndPos);

fbReadBitsFromByte(byData := byActualAppState, iStartBit := 2, iEndBit := 2, byValue => byAdvancedEndPos); 
xAdvancedEndPos_optional :=  BYTE_TO_BIT(byAdvancedEndPos);

fbReadBitsFromByte(byData := byActualAppState, iStartBit := 7, iEndBit := 7, byValue => byWarning);
xWarning := BYTE_TO_BIT(byWarning);

END_FUNCTION_BLOCK

// Transfermode/specific_MA_config/FB_Write_config_MA_02
/// This function block can be used to download the configuration of Motion App 2 ("Proportional directional control valve").
/// The specific parameters of this Motion App are the inputs of this FB and can be defined by the user. 
/// The function block uses the transfer mode to write this configuration to the Motion Terminal
/// and indicates the state of the download process.

FUNCTION_BLOCK FB_Write_config_MA_02
VAR_INPUT
	awBusDataFromVTEM 				: ARRAY [0..2] OF WORD;		(* 6 bytes of process data received from the Motion Terminal *)
END_VAR

VAR_IN_OUT
	awBusDataToVTEM 				: ARRAY [0..2] OF WORD; 	(* 6 bytes of process data sent to the Motion Terminal *)
END_VAR
		
VAR_INPUT
	xExecute 						: BOOL; 					(* has to be set to TRUE for a download and to FALSE to reset the function block after a download *)

	iParameterSet					: INT := 1; 				(* the parameter set to be written to, 1 by default *)

	// system parameters
		iInPortRetracted_optional	: INT;						// Sensor port for detection of end position at pressurisation of outlet port 2 (retracted), value is number of the slot (beginning from 0 and including valve slots) * 10 + number of the port
		iInPortAdvanced_optional	: INT;						// Sensor port for detection of end position at pressurisation of outlet port 4 (advanced), value is number of the slot (beginning from 0 and including valve slots) * 10 + number of the port
	
	// application parameters
		iCharacteristicAt2 			: INT := 0; 				// characteristic of the control algorithm for outlet port 2 (0 = precise, 1 = universal, 2 = fast)
		iCharacteristicAt4 			: INT := 0; 				// characteristic of the control algorithm for outlet port 4 (0 = precise, 1 = universal, 2 = fast)
		iOperatingMode				: INT := 0;	 				// Switching the operating mode (0 = seal seat behaviour, 1 = servo mode)

END_VAR                     		

VAR_OUTPUT                  		
	iResponse 						: eTransferResponse; 		(* returns the status of the execution of the download process *)
	sCurrentValue 					: STRING; 					(* indicates which value of the array is currently treated (necessary to evaluate in case of error messages) *)
	xDownloadDone 					: BOOL; 					(* indicates whether the download was successful *)
	xDownloadError 					: BOOL := FALSE; 			(* indicates whether an error occurred during the transfer *)
END_VAR

VAR
	aTransferPackages				: ARRAY [0..100] OF stTransferPackage;
	fbdownloadMultipleParameters	: FB_Download_Multiple_Parameters;
	iCurrentValue					: INT;
	fbWriteValueToWord 				: FB_Write_Value_To_Word;
END_VAR

(*****************************************************************************************************

Festo SE & Co. KG, Esslingen
Copyright (c) 2021. All rights reserved.

Product:            Motion Terminal VTEM
Description:        Function block to download the parameters for Motion App 2 to the Motion Terminal

Object version:     2.01
Last change:        2021-07
======================================================================================================
                                       H I S T O R Y
======================================================================================================
Version:            2.01
Date:               2021-07
Change/Activity:    - added application parameter iOperatingMode (#4381180)
Release:            3.5.7.237 (CODESYS 3.5.7.2, Lib version 3.7)
Author:             JEBU
------------------------------------------------------------------------------------------------------
Version:            2.00
Date:               2019-03
Change/Activity:    - added parameters for the sensor port mapping (#2256294)
					- changed awBusDataToVTEM into VAR_IN_OUT (#2368965)
Release:            3.5.7.230 (CODESYS 3.5.7.2, Lib version 3.0)
Author:             JEBU
------------------------------------------------------------------------------------------------------
Version:            1.00
Date:               2017
Change/Activity:    - created
Release:            3.5.7.220
Author:             HLBG
======================================================================================================

*****************************************************************************************************)

// write the Motion App specific parameters into the struct
	//iCharacteristicAt2
		aTransferPackages[0].iChannel := iParameterSet;
		aTransferPackages[0].iAddressedTarget := 2;
		aTransferPackages[0].iIndex := 220;
		aTransferPackages[0].iTransferValue := iCharacteristicAt2;
	
	//iCharacteristicAt4
		aTransferPackages[1].iChannel := iParameterSet;
		aTransferPackages[1].iAddressedTarget := 2;
		aTransferPackages[1].iIndex := 221;
		aTransferPackages[1].iTransferValue := iCharacteristicAt4;
	
	//iInPortRetract_optional
		aTransferPackages[2].iChannel := iParameterSet;
		aTransferPackages[2].iAddressedTarget := 2;
		aTransferPackages[2].iIndex := 70;
		aTransferPackages[2].iTransferValue := iInPortRetracted_optional;
	
	//iInPortAdvanced_optional
		aTransferPackages[3].iChannel := iParameterSet;
		aTransferPackages[3].iAddressedTarget := 2;
		aTransferPackages[3].iIndex := 71;
		aTransferPackages[3].iTransferValue := iInPortAdvanced_optional;

	//iOperatingMode
		aTransferPackages[4].iChannel := iParameterSet;
		aTransferPackages[4].iAddressedTarget := 2;
		aTransferPackages[4].iIndex := 223;
		aTransferPackages[4].iTransferValue := iOperatingMode;
	
	// define end of parameter list to be downloaded by setting all variables to 0 (end criterion for FB_Download_Multiple_Parameters)
		aTransferPackages[5].iChannel := 0;
		aTransferPackages[5].iAddressedTarget := 0;
		aTransferPackages[5].iIndex := 0;
		aTransferPackages[5].iTransferValue := 0;


// pre-check of the value for the parameter set
	IF xExecute = TRUE AND (iParameterSet < 1 OR iParameterSet > 5) THEN		// invalid input for the parameter set
		xDownloadDone := FALSE; 
		xDownloadError := TRUE; 
		iResponse := eTransferResponse.invalid_ParameterSet; 
		iCurrentValue := 0; 
		// send command 'stop'
		fbWriteValueToWord(iValue := 61, iStartBit := 0, iEndBit := 5, wDataWord := awBusDataToVTEM[0]); 			// ValveMode = 61
		fbWriteValueToWord(iValue := 0, iStartBit := 6, iEndBit := 15, wDataWord := awBusDataToVTEM[0]); 			// (empty)
		awBusDataToVTEM[1] := 0; 
		awBusDataToVTEM[2] := 0; 
		
	ELSE	
		// call the function block for multiple parameter download
		fbdownloadMultipleParameters(	xExecute := xExecute,
										awBusDataFromVTEM := awBusDataFromVTEM,
										aTransferPackages := aTransferPackages, 
										awBusDataToVTEM := awBusDataToVTEM,
										xDownloadDone => xDownloadDone,
										xDownloadError => xDownloadError,
										iResponse => iResponse,
										iCurrentValue => iCurrentValue);
	END_IF


// The current value output is needed if there is any invalid value in order to address it correctly.
// As the user doesn't work with indices in this function block, the current value is transformed to a string holding the name of the parameter.
	CASE iCurrentValue OF
		0: sCurrentValue := 'iCharacteristicAt2';
		1: sCurrentValue := 'iCharacteristicAt4';
		2: sCurrentValue := 'iInPortRetract_optional';
		3: sCurrentValue := 'iInPortAdvanced_optional';
		4: sCurrentValue := 'iOperatingMode';
		5: sCurrentValue := 'AllParametersWritten';
	END_CASE

END_FUNCTION_BLOCK

// Transfermode/specific_MA_config/FB_Write_config_MA_03
/// This function block can be used to download the configuration of Motion App 3 ("Proportional pressure regulation").
/// The specific parameters of this Motion App are the inputs of this FB and can be defined by the user. 
/// The function block uses the transfer mode to write this configuration to the Motion Terminal
/// and indicates the state of the download process.

FUNCTION_BLOCK FB_Write_config_MA_03
VAR_INPUT
	awBusDataFromVTEM 				: ARRAY [0..2] OF WORD;		(* 6 bytes of process data received from the Motion Terminal *)
END_VAR	

VAR_IN_OUT
	awBusDataToVTEM 				: ARRAY [0..2] OF WORD; 	(* 6 bytes of process data sent to the Motion Terminal *)
END_VAR

VAR_INPUT
	xExecute 						: BOOL; 					(* has to be set to TRUE for a download and to FALSE to reset the function block after a download *)
		                    		
	iParameterSet					: INT := 1; 				(* the parameter set to be written to, 1 by default *)
	
	// system parameters
		iInPortRetracted_optional	: INT;						// Sensor port for detection of end position at pressurisation of outlet port 2 (retracted), value is number of the slot (beginning from 0 and including valve slots) * 10 + number of the port
		iInPortAdvanced_optional	: INT;						// Sensor port for detection of end position at pressurisation of outlet port 4 (advanced), value is number of the slot (beginning from 0 and including valve slots) * 10 + number of the port
	
	// application parameters
		iCharacteristicAt2 			: INT;		 				// characteristic of the control algorithm for outlet port 2 (0 = small volumes ≥0.05 l … ≤0.1 l, 1 = medium volumes >0.1 l … <1.0 l, 2 = large volumes ≥1.0 l, 3 = customized characteristic defined by tuning parameters)
		iCharacteristicAt4 			: INT; 						// characteristic of the control algorithm for outlet port 4 (0 = small volumes ≥0.05 l … ≤0.1 l, 1 = medium volumes >0.1 l … <1.0 l, 2 = large volumes ≥1.0 l, 3 = customized characteristic defined by tuning parameters)

	//tuning parameters
		iOptProportionalGainFor2	: INT;						// Optional tuning parameter for the customized proportional element of the PID modulator at outlet port 2 [1 digit = 0.01 g/s/bar]
		iOptIntegralGainFor2		: INT;						// Optional tuning parameter for the customized integral element of the PID modulator at outlet port 2 [1 digit = 0.01 g/s²/bar]
		iOptTimeConstantFor2		: INT;						// Optional tuning parameter for the customized time constant element of the PID modulator at outlet port 2 [1 digit = 0.001 s]
		iOptShiftZeroPointSwitchOff2	: INT;					// Optional tuning parameter for shifting the zero point switch-off for outlet port 2 [1 digit = 0.001 bar]
		iOptProportionalGainFor4	: INT;						// Optional tuning parameter for the customized proportional element of the PID modulator at outlet port 4 [1 digit = 0.01 g/s/bar]
		iOptIntegralGainFor4		: INT;						// Optional tuning parameter for the customized integral element of the PID modulator at outlet port 4 [1 digit = 0.01 g/s²/bar]
		iOptTimeConstantFor4		: INT;						// Optional tuning parameter for the customized time constant element of the PID modulator at outlet port 4 [1 digit = 0.001 s]
		iOptShiftZeroPointSwitchOff4	: INT;					// Optional tuning parameter for shifting the zero point switch-off for outlet port 4 [1 digit = 0.001 bar]
END_VAR                     		

VAR_OUTPUT                  		
	iResponse 						: eTransferResponse; 		(* returns the status of the execution of the download process *)
	sCurrentValue 					: STRING; 					(* indicates which value of the array is currently treated (necessary to evaluate in case of error messages) *)
	xDownloadDone 					: BOOL; 					(* indicates whether the download was successful *)
	xDownloadError 					: BOOL := FALSE; 			(* indicates whether an error occurred during the transfer *)
END_VAR                     		

VAR                         		
	aTransferPackages				: ARRAY [0..100] OF stTransferPackage;
	fbdownloadMultipleParameters	: FB_Download_Multiple_Parameters;
	iCurrentValue					: INT;
	fbWriteValueToWord 				: FB_Write_Value_To_Word;
END_VAR

(*****************************************************************************************************

Festo SE & Co. KG, Esslingen
Copyright (c) 2018. All rights reserved.

Product:            Motion Terminal VTEM
Description:        Function block to download the parameters for Motion App 3 to the Motion Terminal

Object version:     2.01
Last change:        2020-11
======================================================================================================
                                       H I S T O R Y
======================================================================================================
Version:            2.01
Date:               2020-11
Change/Activity:    - added tuning parameters for zero point switch-off (#3800154)
Release:            3.5.7.236 (CODESYS 3.5.7.2, Lib version 3.6)
Author:             JEBU
------------------------------------------------------------------------------------------------------
Version:            2.00
Date:               2019-03
Change/Activity:    - added parameters for the sensor port mapping (#2256294)
                    - changed awBusDataToVTEM into VAR_IN_OUT (#2368965)
Release:            3.5.7.230 (CODESYS 3.5.7.2, Lib version 3.0)
Author:             JEBU
------------------------------------------------------------------------------------------------------
Version:            1.01
Date:               2018-11
Change/Activity:    - added tuning parameters (#2257307)
Release:            3.5.7.221
Author:             JEBU
------------------------------------------------------------------------------------------------------
Version:            1.00
Date:               2017
Change/Activity:    - created
Release:            3.5.7.220
Author:             HLBG
======================================================================================================

*****************************************************************************************************)

// write the Motion App specific parameters into the struct
	//iCharacteristicAt2
		aTransferPackages[0].iChannel := iParameterSet;
		aTransferPackages[0].iAddressedTarget := 3;
		aTransferPackages[0].iIndex := 220;
		aTransferPackages[0].iTransferValue := iCharacteristicAt2;
	
	//iCharacteristicAt4
		aTransferPackages[1].iChannel := iParameterSet;
		aTransferPackages[1].iAddressedTarget := 3;
		aTransferPackages[1].iIndex := 221;
		aTransferPackages[1].iTransferValue := iCharacteristicAt4;
	
	//iOptProportionalGainFor2
		aTransferPackages[2].iChannel := iParameterSet;
		aTransferPackages[2].iAddressedTarget := 3;
		aTransferPackages[2].iIndex := 230;
		aTransferPackages[2].iTransferValue := iOptProportionalGainFor2;
		
	//iOptIntegralGainFor2
		aTransferPackages[3].iChannel := iParameterSet;
		aTransferPackages[3].iAddressedTarget := 3;
		aTransferPackages[3].iIndex := 231;
		aTransferPackages[3].iTransferValue := iOptIntegralGainFor2;
		
	//iOptTimeConstantFor2
		aTransferPackages[4].iChannel := iParameterSet;
		aTransferPackages[4].iAddressedTarget := 3;
		aTransferPackages[4].iIndex := 232;
		aTransferPackages[4].iTransferValue := iOptTimeConstantFor2;

	//iOptShiftZeroPointSwitchOff2
		aTransferPackages[5].iChannel := iParameterSet;
		aTransferPackages[5].iAddressedTarget := 3;
		aTransferPackages[5].iIndex := 233;
		aTransferPackages[5].iTransferValue := iOptShiftZeroPointSwitchOff2;
		
	//iOptProportionalGainFor4
		aTransferPackages[6].iChannel := iParameterSet;
		aTransferPackages[6].iAddressedTarget := 3;
		aTransferPackages[6].iIndex := 240;
		aTransferPackages[6].iTransferValue := iOptProportionalGainFor4;
		
	//iOptIntegralGainFor4
		aTransferPackages[7].iChannel := iParameterSet;
		aTransferPackages[7].iAddressedTarget := 3;
		aTransferPackages[7].iIndex := 241;
		aTransferPackages[7].iTransferValue := iOptIntegralGainFor4;
		
	//iOptTimeConstantFor4
		aTransferPackages[8].iChannel := iParameterSet;
		aTransferPackages[8].iAddressedTarget := 3;
		aTransferPackages[8].iIndex := 242;
		aTransferPackages[8].iTransferValue := iOptTimeConstantFor4;
	
	//iOptShiftZeroPointSwitchOff4
		aTransferPackages[9].iChannel := iParameterSet;
		aTransferPackages[9].iAddressedTarget := 3;
		aTransferPackages[9].iIndex := 243;
		aTransferPackages[9].iTransferValue := iOptShiftZeroPointSwitchOff4;

	//iInPortRetract_optional
		aTransferPackages[10].iChannel := iParameterSet;
		aTransferPackages[10].iAddressedTarget := 3;
		aTransferPackages[10].iIndex := 70;
		aTransferPackages[10].iTransferValue := iInPortRetracted_optional;
	
	//iInPortAdvanced_optional
		aTransferPackages[11].iChannel := iParameterSet;
		aTransferPackages[11].iAddressedTarget := 3;
		aTransferPackages[11].iIndex := 71;
		aTransferPackages[11].iTransferValue := iInPortAdvanced_optional;
		
	// define end of parameter list to be downloaded by setting all variables to 0 (end criterion for FB_Download_Multiple_Parameters)
		aTransferPackages[12].iChannel := 0;
		aTransferPackages[12].iAddressedTarget := 0;
		aTransferPackages[12].iIndex := 0;
		aTransferPackages[12].iTransferValue := 0;

// pre-check of the value for the parameter set
	IF xExecute = TRUE AND (iParameterSet < 1 OR iParameterSet > 5) THEN		// invalid input for the parameter set
		xDownloadDone := FALSE; 
		xDownloadError := TRUE; 
		iResponse := eTransferResponse.invalid_ParameterSet; 
		iCurrentValue := 0; 
		// send command 'stop'
		fbWriteValueToWord(iValue := 61, iStartBit := 0, iEndBit := 5, wDataWord := awBusDataToVTEM[0]); 			// ValveMode = 61
		fbWriteValueToWord(iValue := 0, iStartBit := 6, iEndBit := 15, wDataWord := awBusDataToVTEM[0]); 			// (empty)
		awBusDataToVTEM[1] := 0; 
		awBusDataToVTEM[2] := 0; 
		
	ELSE	
		// call the function block for multiple parameter download
			fbdownloadMultipleParameters(	xExecute := xExecute,
											awBusDataFromVTEM := awBusDataFromVTEM,
											aTransferPackages := aTransferPackages, 
											awBusDataToVTEM := awBusDataToVTEM,
											xDownloadDone => xDownloadDone,
											xDownloadError => xDownloadError,
											iResponse => iResponse,
											iCurrentValue => iCurrentValue);
	END_IF

// The current value output is needed if there is any invalid value in order to address it correctly.
// As the user doesn't work with indices in this function block, the current value is transformed to a string holding the name of the parameter.
	CASE iCurrentValue OF
		0: sCurrentValue := 'iCharacteristicAt2';
		1: sCurrentValue := 'iCharacteristicAt4';
		2: sCurrentValue := 'iOptProportionalGainFor2';
		3: sCurrentValue := 'iOptIntegralGainFor2';
		4: sCurrentValue := 'iOptTimeConstantFor2';
		5: sCurrentValue := 'iOptShiftZeroPointSwitchOff2';
		6: sCurrentValue := 'iOptProportionalGainFor4';
		7: sCurrentValue := 'iOptIntegralGainFor4';
		8: sCurrentValue := 'iOptTimeConstantFor4';
		9: sCurrentValue := 'iOptShiftZeroPointSwitchOff4';
		10: sCurrentValue := 'iInPortRetract_optional';
		11: sCurrentValue := 'iInPortAdvanced_optional';
		12: sCurrentValue := 'AllParametersWritten';
	END_CASE

END_FUNCTION_BLOCK

// Transfermode/specific_MA_config/FB_Write_config_MA_08
/// This function block can be used to download the configuration of Motion App 8 ("Selectable pressure level (ECO)").
/// The specific parameters of this Motion App are the inputs of this FB and can be defined by the user. 
/// The function block uses the transfer mode to write this configuration to the Motion Terminal
/// and indicates the state of the download process.

FUNCTION_BLOCK FB_Write_config_MA_08
VAR_INPUT
	awBusDataFromVTEM 				: ARRAY [0..2] OF WORD;		(* 6 bytes of process data received from the Motion Terminal *)
END_VAR

VAR_IN_OUT
	awBusDataToVTEM 				: ARRAY [0..2] OF WORD; 	(* 6 bytes of process data sent to the Motion Terminal *)
END_VAR

VAR_INPUT
	xExecute 						: BOOL; 					(* has to be set to TRUE for a download and to FALSE to reset the function block after a download *)
		                    		                        	
	iParameterSet					: INT := 1; 				(* the parameter set to be written to, 1 by default *)
	
	// system parameters
		iTubingLengthAt2 			: INT; 						(* length of the tubing connected to outlet port 2 of the valve [1 digit = 1 mm] *)
	 	iTubingLengthAt4 			: INT;						(* length of the tubing connected to outlet port 4 of the valve [1 digit = 1 mm] *)
	 	iTubingInnerDiameterAt2		: INT;  					(* inner diameter of the tubing connected to outlet port 2 of the valve [1 digit = 0.01 mm] *)
	 	iTubingInnerDiameterAt4		: INT;						(* inner diameter of the tubing connected to outlet port 4 of the valve [1 digit = 0.01 mm] *)
	 	iDriveType 					: INT;						// type of the drive/cylinder/... that is to be operated by the valve ->  see list of drive types at support portal (www.festo.com/sp/)
	 	iDriveStroke 				: INT; 						(* stroke of the drive/cylinder/... that is to be operated by the valve [1 digit = 1 mm for linear drives, 1 digit = 1° for rotary drives] *)
		iInstallationPositionDrive 	: INT;  	 				(* inclination of the cylinder with reference to a horizontal installation position [1 digit = 0.01°, positive values = advancing upwards] *)
		iInPortRetracted_optional	: INT;						// Sensor port for detection of end position at pressurisation of outlet port 2 (retracted), value is number of the slot (beginning from 0 and including valve slots) * 10 + number of the port
		iInPortAdvanced_optional	: INT;						// Sensor port for detection of end position at pressurisation of outlet port 4 (advanced), value is number of the slot (beginning from 0 and including valve slots) * 10 + number of the port
	
	// application parameters                               	
		iLoadRetracting 			: INT;						(* mass that is to be moved by the drive when retracting ((2) pressurised) [1 digit = 0.01 kg] *)
	 	iLoadAdvancing 				: INT; 						(* mass that is to be moved by the drive when advancing ((4) pressurised) [1 digit = 0.01 kg] *)
		iMomentOfInertiaRetracting	: INT;						// Moment of inertia during for swivel drives when retratcting ((2) pressirised) [1 digit = 1 kg cm³]
		iMomentOfInertiaAdvancing	: INT;						// Moment of inertia during for swivel drives when advancing ((4) pressirised) [1 digit = 1 kg cm³]
		iSoftStartFunction			: INT := 1;					(* flag to enable or disable the iSoftStartFunction; 0 = disabled, 1 = enabled *)
	
	//tuning parameters
		iOptProportionalGainFor2	: INT;						// Optional tuning parameter for the customized proportional element of the PID modulator at outlet port 2 [1 digit = 1 %]
		iOptProportionalGainFor4	: INT;						// Optional tuning parameter for the customized proportional element of the PID modulator at outlet port 4 [1 digit = 1 %]
END_VAR

VAR_OUTPUT                                                  	
	iResponse 						: eTransferResponse; 		(* returns the status of the execution of the download process *)
	sCurrentValue 					: STRING; 					(* indicates which value of the array is currently treated (necessary to evaluate in case of error messages) *)
	xDownloadDone 					: BOOL; 					(* indicates whether the download was successful *)
	xDownloadError 					: BOOL := FALSE; 			(* indicates whether an error occurred during the transfer *)
END_VAR

VAR
	aTransferPackages				: ARRAY [0..100] OF stTransferPackage;
	fbdownloadMultipleParameters 	: FB_Download_Multiple_Parameters;
	iCurrentValue					: INT;
	fbWriteValueToWord 				: FB_Write_Value_To_Word;
END_VAR

(*****************************************************************************************************

Festo SE & Co. KG, Esslingen
Copyright (c) 2021. All rights reserved.

Product:            Motion Terminal VTEM
Description:        Function block to download the parameters for Motion App 8 to the Motion Terminal

Object version:     2.01
Last change:        2021-08
======================================================================================================
                                       H I S T O R Y
======================================================================================================
Version:            2.01
Date:               2021-08
Change/Activity:    - added tuning parameters (#4510538)
Release:            3.5.7.237 (CODESYS 3.5.7.2, Lib version 3.7)
Author:             JEBU
------------------------------------------------------------------------------------------------------
Version:            2.00
Date:               2019-03
Change/Activity:    - added parameters for moment of inertia used for swivel drives (#2307852)
                    - added parameters for the sensor port mapping (#2256294)
                    - changed awBusDataToVTEM into VAR_IN_OUT (#2368965)
Release:            3.5.7.230 (CODESYS 3.5.7.2, Lib version 3.0)
Author:             JEBU
------------------------------------------------------------------------------------------------------
Version:            1.00
Date:               2017
Change/Activity:    - created
Release:            3.5.7.220
Author:             HLBG
======================================================================================================

*****************************************************************************************************)

// write the Motion App specific parameters into the struct
	//iTubingLengthAt2
		aTransferPackages[0].iChannel := iParameterSet;
		aTransferPackages[0].iAddressedTarget := 8;
		aTransferPackages[0].iIndex := 12;
		aTransferPackages[0].iTransferValue := iTubingLengthAt2;
		
	//iTubingLengthAt4
		aTransferPackages[1].iChannel := iParameterSet;
		aTransferPackages[1].iAddressedTarget := 8;
		aTransferPackages[1].iIndex := 13;
		aTransferPackages[1].iTransferValue := iTubingLengthAt4;
		
	//iTubingInnerDiameterAt2
		aTransferPackages[2].iChannel := iParameterSet;
		aTransferPackages[2].iAddressedTarget := 8;
		aTransferPackages[2].iIndex := 14;
		aTransferPackages[2].iTransferValue := iTubingInnerDiameterAt2;
		
	//iTubingInnerDiameterAt4
		aTransferPackages[3].iChannel := iParameterSet;
		aTransferPackages[3].iAddressedTarget := 8;
		aTransferPackages[3].iIndex := 15;
		aTransferPackages[3].iTransferValue := iTubingInnerDiameterAt4;
		
	//iDriveType
		aTransferPackages[4].iChannel := iParameterSet;
		aTransferPackages[4].iAddressedTarget := 8;
		aTransferPackages[4].iIndex := 20;
		aTransferPackages[4].iTransferValue := iDriveType;
		
	//iDriveStroke
		aTransferPackages[5].iChannel := iParameterSet;
		aTransferPackages[5].iAddressedTarget := 8;
		aTransferPackages[5].iIndex := 21;
		aTransferPackages[5].iTransferValue := iDriveStroke;
		
	//iInstallationPositionDrive
		aTransferPackages[6].iChannel := iParameterSet;
		aTransferPackages[6].iAddressedTarget := 8;
		aTransferPackages[6].iIndex := 60;
		aTransferPackages[6].iTransferValue := iInstallationPositionDrive;
		
	//iLoadRetracting
		aTransferPackages[7].iChannel := iParameterSet;
		aTransferPackages[7].iAddressedTarget := 8;
		aTransferPackages[7].iIndex := 100;
		aTransferPackages[7].iTransferValue := iLoadRetracting;
		
	//iLoadAdvancing
		aTransferPackages[8].iChannel := iParameterSet;
		aTransferPackages[8].iAddressedTarget := 8;
		aTransferPackages[8].iIndex := 101;
		aTransferPackages[8].iTransferValue := iLoadAdvancing;
		
	//iMomentOfInertiaRetracting
		aTransferPackages[9].iChannel := iParameterSet;
		aTransferPackages[9].iAddressedTarget := 8;
		aTransferPackages[9].iIndex := 102;
		aTransferPackages[9].iTransferValue := iMomentOfInertiaRetracting;
	
	//iMomentOfInertiaAdvancing
		aTransferPackages[10].iChannel := iParameterSet;
		aTransferPackages[10].iAddressedTarget := 8;
		aTransferPackages[10].iIndex := 103;
		aTransferPackages[10].iTransferValue := iMomentOfInertiaAdvancing;

	//iSoftStartFunction
		aTransferPackages[11].iChannel := iParameterSet;
		aTransferPackages[11].iAddressedTarget := 8;
		aTransferPackages[11].iIndex := 222;
		aTransferPackages[11].iTransferValue := iSoftStartFunction;
		
	//iInPortRetract_optional
		aTransferPackages[12].iChannel := iParameterSet;
		aTransferPackages[12].iAddressedTarget := 8;
		aTransferPackages[12].iIndex := 70;
		aTransferPackages[12].iTransferValue := iInPortRetracted_optional;
	
	//iInPortAdvanced_optional
		aTransferPackages[13].iChannel := iParameterSet;
		aTransferPackages[13].iAddressedTarget := 8;
		aTransferPackages[13].iIndex := 71;
		aTransferPackages[13].iTransferValue := iInPortAdvanced_optional;
	
	//iOptProportionalGainFor2
		aTransferPackages[14].iChannel := iParameterSet;
		aTransferPackages[14].iAddressedTarget := 8;
		aTransferPackages[14].iIndex := 239;
		aTransferPackages[14].iTransferValue := iOptProportionalGainFor2;
	
	//iOptProportionalGainFor4
		aTransferPackages[15].iChannel := iParameterSet;
		aTransferPackages[15].iAddressedTarget := 8;
		aTransferPackages[15].iIndex := 249;
		aTransferPackages[15].iTransferValue := iOptProportionalGainFor4;
	
	// define end of parameter list to be downloaded by setting all variables to 0 (end criterion for FB_Download_Multiple_Parameters)
		aTransferPackages[16].iChannel := 0;
		aTransferPackages[16].iAddressedTarget := 0;
		aTransferPackages[16].iIndex := 0;
		aTransferPackages[16].iTransferValue := 0;


// pre-check of the value for the parameter set
	IF xExecute = TRUE AND (iParameterSet < 1 OR iParameterSet > 5) THEN		// invalid input for the parameter set
		xDownloadDone := FALSE; 
		xDownloadError := TRUE; 
		iResponse := eTransferResponse.invalid_ParameterSet; 
		iCurrentValue := 0; 
		// send command 'stop'
		fbWriteValueToWord(iValue := 61, iStartBit := 0, iEndBit := 5, wDataWord := awBusDataToVTEM[0]); 			// ValveMode = 61
		fbWriteValueToWord(iValue := 0, iStartBit := 6, iEndBit := 15, wDataWord := awBusDataToVTEM[0]); 			// (empty)
		awBusDataToVTEM[1] := 0; 
		awBusDataToVTEM[2] := 0; 
		
	ELSE	
		// call the function block for multiple parameter download
			fbdownloadMultipleParameters(	xExecute := xExecute,
											awBusDataFromVTEM := awBusDataFromVTEM,
											aTransferPackages := aTransferPackages, 
											awBusDataToVTEM := awBusDataToVTEM,
											xDownloadDone => xDownloadDone,
											xDownloadError => xDownloadError,
											iResponse => iResponse,
											iCurrentValue => iCurrentValue);
	END_IF


// The current value output is needed if there is any invalid value in order to address it correctly.
// As the user doesn't work with indices in this function block, the current value is transformed to a string holding the name of the parameter.
	CASE iCurrentValue OF
		0: sCurrentValue := 'iTubingLengthAt2';
		1: sCurrentValue := 'iTubingLengthAt4';
		2: sCurrentValue := 'iTubingInnerDiameterAt2';
		3: sCurrentValue := 'iTubingInnerDiameterAt4';
		4: sCurrentValue := 'iDriveType';
		5: sCurrentValue := 'iDriveStroke';
		6: sCurrentValue := 'iInstallationPositionDrive';
		7: sCurrentValue := 'iLoadRetracting';
		8: sCurrentValue := 'iLoadAdvancing';
		9: sCurrentValue := 'iMomentOfInertiaRetracting';
		10: sCurrentValue := 'iMomentOfInertiaAdvancing';
		11: sCurrentValue := 'iSoftStartFunction';
		12: sCurrentValue := 'iInPortRetract_optional';
		13: sCurrentValue := 'iInPortAdvanced_optional';
		14: sCurrentValue := 'iOptProportionalGainFor2';
		15: sCurrentValue := 'iOptProportionalGainFor4';
	  	16: sCurrentValue := 'AllParametersWritten';
	END_CASE

END_FUNCTION_BLOCK

// Transfermode/specific_MA_config/FB_Write_config_MA_05
/// This function block can be used to download the configuration of Motion App 5 ("Supply and exhaust air flow control").
/// The specific parameters of this Motion App are the inputs of this FB and can be defined by the user. 
/// The function block uses the transfer mode to write this configuration to the Motion Terminal
/// and indicates the state of the download process.

FUNCTION_BLOCK FB_Write_config_MA_05
VAR_INPUT
	awBusDataFromVTEM 				: ARRAY [0..2] OF WORD;		(* 6 bytes of process data received from the Motion Terminal *)
END_VAR

VAR_IN_OUT
	awBusDataToVTEM 				: ARRAY [0..2] OF WORD; 	(* 6 bytes of process data sent to the Motion Terminal *)
END_VAR

VAR_INPUT
	xExecute 						: BOOL; 					(* has to be set to TRUE for a download and to FALSE to reset the function block after a download *)
		                    		                        		
	iParameterSet					: INT := 1; 				(* the parameter set to be written to, 1 by default *)
                                                    		
	// system parameters
		iInPortRetracted_optional	: INT;						// Sensor port for detection of end position at pressurisation of outlet port 2 (retracted), value is number of the slot (beginning from 0 and including valve slots) * 10 + number of the port
		iInPortAdvanced_optional	: INT;						// Sensor port for detection of end position at pressurisation of outlet port 4 (advanced), value is number of the slot (beginning from 0 and including valve slots) * 10 + number of the port

	// application parameters                       	
		iSoftStartFunction			: INT := 1;					(* flag to enable or disable the SoftStartFunction; 0 = disabled, 1 = enabled *)
END_VAR

VAR_OUTPUT
	iResponse 						: eTransferResponse; 		(* returns the status of the execution of the download process *)
	sCurrentValue 					: STRING; 					(* indicates which value of the array is currently treated (necessary to evaluate in case of error messages) *)
	xDownloadDone 					: BOOL; 					(* indicates whether the download was successful *)
	xDownloadError 					: BOOL := FALSE; 			(* indicates whether an error occurred during the transfer *)
END_VAR

VAR
	aTransferPackages				: ARRAY [0..100] OF stTransferPackage; 
	fbdownloadMultipleParameters 	: FB_Download_Multiple_Parameters; 
	iCurrentValue					: INT;
	fbWriteValueToWord 				: FB_Write_Value_To_Word; 
END_VAR

(*****************************************************************************************************

Festo SE & Co. KG, Esslingen
Copyright (c) 2018. All rights reserved.

Product:            Motion Terminal VTEM
Description:        Function block to download the parameters for Motion App 5 to the Motion Terminal

Object version:     2.00
Last change:        2019-03
======================================================================================================
                                       H I S T O R Y
======================================================================================================
Version:            2.00
Date:               2019-03
Change/Activity:    - added parameters for the sensor port mapping (#2256294)
                    - changed awBusDataToVTEM into VAR_IN_OUT (#2368965)
Release:            3.5.7.230 (CODESYS 3.5.7.2, Lib version 3.0)
Author:             JEBU
------------------------------------------------------------------------------------------------------
Version:            1.00
Date:               2017
Change/Activity:    - created
Release:            3.5.7.220
Author:             HLBG
======================================================================================================

*****************************************************************************************************)

// write the Motion App specific parameters into the struct
	//iSoftStartFunction
		aTransferPackages[0].iChannel := iParameterSet;
		aTransferPackages[0].iAddressedTarget := 5;
		aTransferPackages[0].iIndex := 222;
		aTransferPackages[0].iTransferValue := iSoftStartFunction;
	
	//iInPortRetract_optional
		aTransferPackages[1].iChannel := iParameterSet;
		aTransferPackages[1].iAddressedTarget := 5;
		aTransferPackages[1].iIndex := 70;
		aTransferPackages[1].iTransferValue := iInPortRetracted_optional;
	
	//iInPortAdvanced_optional
		aTransferPackages[2].iChannel := iParameterSet;
		aTransferPackages[2].iAddressedTarget := 5;
		aTransferPackages[2].iIndex := 71;
		aTransferPackages[2].iTransferValue := iInPortAdvanced_optional;
	
	// define end of parameter list to be downloaded by setting all variables to 0 (end criterion for FB_Download_Multiple_Parameters)
		aTransferPackages[3].iChannel := 0;
		aTransferPackages[3].iAddressedTarget := 0;
		aTransferPackages[3].iIndex := 0;
		aTransferPackages[3].iTransferValue := 0;


// pre-check of the value for the parameter set
	IF xExecute = TRUE AND (iParameterSet < 1 OR iParameterSet > 5) THEN		// invalid input for the parameter set
		xDownloadDone := FALSE; 
		xDownloadError := TRUE; 
		iResponse := eTransferResponse.invalid_ParameterSet; 
		iCurrentValue := 0; 
		// send command 'stop'
		fbWriteValueToWord(iValue := 61, iStartBit := 0, iEndBit := 5, wDataWord := awBusDataToVTEM[0]); 			// ValveMode = 61
		fbWriteValueToWord(iValue := 0, iStartBit := 6, iEndBit := 15, wDataWord := awBusDataToVTEM[0]); 			// (empty)
		awBusDataToVTEM[1] := 0; 
		awBusDataToVTEM[2] := 0; 
		
	ELSE	
		// call the function block for multiple parameter download
			fbdownloadMultipleParameters(	xExecute := xExecute,
											awBusDataFromVTEM := awBusDataFromVTEM,
											aTransferPackages := aTransferPackages, 
											awBusDataToVTEM := awBusDataToVTEM,
											xDownloadDone => xDownloadDone,
											xDownloadError => xDownloadError,
											iResponse => iResponse,
											iCurrentValue => iCurrentValue);
	END_IF


// The current value output is needed if there is any invalid value in order to address it correctly.
// As the user doesn't work with indices in this function block, the current value is transformed to a string holding the name of the parameter.
	CASE iCurrentValue OF
		0: sCurrentValue := 'iSoftStartFunction';
		1: sCurrentValue := 'iInPortRetract_optional';
		2: sCurrentValue := 'iInPortAdvanced_optional';
		3: sCurrentValue := 'AllParametersWritten';
	END_CASE

END_FUNCTION_BLOCK

// StateInterpreter/FB_StateInterpreter_MA_33
/// The variable "byActualAppState" is an output of the FB_ValveControl that is used differently in each Motion App.
/// This function block interprets the "AppState" output of the FB_ValveControl if Motion App 33 ("Positioning") is running.
/// The Motion App specific values are derived from the "byActualAppState".

FUNCTION_BLOCK FB_StateInterpreter_MA_33
VAR_INPUT
	byActualAppState 			: BYTE; 	// output of the FB_ValveControl
END_VAR
VAR_OUTPUT
	xRetractedEndPos			: BOOL;  	// indicates whether the retracted end position (outlet port 4 pressurised) was reached (<= 1 mm) 
	xAdvancedEndPos				: BOOL;  	// indicates whether the advanced end position (outlet port 4 pressurised) was reached (<= 1 mm) 
	xTargetPositionReached		: BOOL;  	// TRUE if the absolute deviation of the actual position from the setpoint position does not exceed the value defined in the "Tolerance for Target Position Reached" parameter for at least the duration defined in the "Damping time for Target Position Reached" parameter.  
	xOvershootInPlannedPath		: BOOL;		// TRUE if the planned path contains an overshoot over the target position
	xControlledStop				: BOOL;		// TRUE if a controlled stop was triggered by an end position violation (only active if the end position monitoring was not deactivated by the corresponding application parameter)
	xWarning					: BOOL; 	// indicates whether there is a warning returned by the Motion App
END_VAR
VAR
	fbReadBitsFromByte			: FB_Read_Bits_From_Byte;
	byRetractedEndPos			: BYTE;
	byAdvancedEndPos			: BYTE;
	byTargetPositionReached		: BYTE;
	byOvershootInPlannedPath	: BYTE;
	byControlledStop			: BYTE;      
	byWarning					: BYTE;
END_VAR

(*****************************************************************************************************

Festo SE & Co. KG, Esslingen
Copyright (c) 2019. All rights reserved.

Product:            Motion Terminal VTEM
Description:        Function block for interpreting the app state of Motion App 33 

Object version:     1.01
Last change:        2020-04
======================================================================================================
                                       H I S T O R Y
======================================================================================================
Version:            1.01
Date:               2020-04
Change/Activity:    - created (#2256322)
Release:            3.5.7.234
Author:             JEBU
======================================================================================================

*****************************************************************************************************)

// read the Motion App specific values from the ActualAppState byte
fbReadBitsFromByte(byData := byActualAppState, iStartBit := 0, iEndBit := 0, byValue => byRetractedEndPos);
xRetractedEndPos :=  BYTE_TO_BIT(byRetractedEndPos);

fbReadBitsFromByte(byData := byActualAppState, iStartBit := 2, iEndBit := 2, byValue => byAdvancedEndPos); 
xAdvancedEndPos :=  BYTE_TO_BIT(byAdvancedEndPos);

fbReadBitsFromByte(byData := byActualAppState, iStartBit := 1, iEndBit := 1, byValue => byTargetPositionReached);
xTargetPositionReached :=  BYTE_TO_BIT(byTargetPositionReached);

fbReadBitsFromByte(byData := byActualAppState, iStartBit := 5, iEndBit := 5, byValue => byOvershootInPlannedPath);
xOvershootInPlannedPath :=  BYTE_TO_BIT(byOvershootInPlannedPath);

fbReadBitsFromByte(byData := byActualAppState, iStartBit := 6, iEndBit := 6, byValue => byControlledStop);
xControlledStop :=  BYTE_TO_BIT(byControlledStop);

fbReadBitsFromByte(byData := byActualAppState, iStartBit := 7, iEndBit := 7, byValue => byWarning);
xWarning := BYTE_TO_BIT(byWarning);

END_FUNCTION_BLOCK

// Transfermode/specific_MA_config/FB_Write_config_MA_01
/// This function block can be used to download the configuration of Motion App 1 ("Directional control valve functions").
/// The specific parameters of this Motion App are the inputs of this FB and can be defined by the user. 
/// The function block uses the transfer mode to write this configuration to the Motion Terminal
/// and indicates the state of the download process.

FUNCTION_BLOCK FB_Write_config_MA_01
VAR_INPUT
	awBusDataFromVTEM 				: ARRAY [0..2] OF WORD;		(* 6 bytes of process data received from the Motion Terminal *)
END_VAR
	
VAR_IN_OUT
	awBusDataToVTEM 				: ARRAY [0..2] OF WORD; 	(* 6 bytes of process data sent to the Motion Terminal *)
END_VAR

VAR_INPUT
	xExecute 						: BOOL; 					(* has to be set to TRUE for a download and to FALSE to reset the function block after a download *)

	iParameterSet					: INT := 1; 				(* the parameter set to be written to, 1 by default *)
	
	// system parameters
		iInPortRetracted_optional	: INT;						// Sensor port for detection of end position at pressurisation of outlet port 2 (retracted), value is number of the slot (beginning from 0 and including valve slots) * 10 + number of the port
		iInPortAdvanced_optional	: INT;						// Sensor port for detection of end position at pressurisation of outlet port 4 (advanced), value is number of the slot (beginning from 0 and including valve slots) * 10 + number of the port

	// application parameters
		iOperatingMode				: INT := 0;	 				// Switching the operating mode (0 = open loop controlled, 1 = close-loop controlled) 
END_VAR                     		

VAR_OUTPUT                  		
	iResponse 						: eTransferResponse; 		(* returns the status of the execution of the download process *)
	sCurrentValue 					: STRING; 					(* indicates which value of the array is currently treated (necessary to evaluate in case of error messages) *)
	xDownloadDone 					: BOOL; 					(* indicates whether the download was successful *)
	xDownloadError 					: BOOL := FALSE; 			(* indicates whether an error occurred during the transfer *)
END_VAR

VAR
	aTransferPackages				: ARRAY [0..100] OF stTransferPackage;
	fbdownloadMultipleParameters 	: FB_Download_Multiple_Parameters;
	iCurrentValue					: INT;
	fbWriteValueToWord 				: FB_Write_Value_To_Word;
END_VAR

(*****************************************************************************************************

Festo SE & Co. KG, Esslingen
Copyright (c) 2018. All rights reserved.

Product:            Motion Terminal VTEM
Description:        Function Block to download the parameters for Motion App 1 to the Motion Terminal

Object version:     2.00
Last change:        2019-03
======================================================================================================
                                       H I S T O R Y
======================================================================================================
Version:            2.00
Date:               2019-03
Change/Activity:    - created (#2256983)
Release:            3.5.7.230 (CODESYS 3.5.7.2, Lib version 3.0)
Author:             JEBU
======================================================================================================

*****************************************************************************************************)

// write the Motion App specific parameters into the struct
	//iOperatingMode
		aTransferPackages[0].iChannel := iParameterSet;
		aTransferPackages[0].iAddressedTarget := 1;
		aTransferPackages[0].iIndex := 223;
		aTransferPackages[0].iTransferValue := iOperatingMode;
	
	//iInPortRetract_optional
		aTransferPackages[1].iChannel := iParameterSet;
		aTransferPackages[1].iAddressedTarget := 1;
		aTransferPackages[1].iIndex := 70;
		aTransferPackages[1].iTransferValue := iInPortRetracted_optional;
	
	//iInPortRetract_optional
		aTransferPackages[2].iChannel := iParameterSet;
		aTransferPackages[2].iAddressedTarget := 1;
		aTransferPackages[2].iIndex := 71;
		aTransferPackages[2].iTransferValue := iInPortAdvanced_optional;
	
	// define end of parameter list to be downloaded by setting all variables to 0 (end criterion for FB_Download_Multiple_Parameters)
		aTransferPackages[3].iChannel := 0;
		aTransferPackages[3].iAddressedTarget := 0;
		aTransferPackages[3].iIndex := 0;
		aTransferPackages[3].iTransferValue := 0;


// pre-check of the value for the parameter set
	IF xExecute = TRUE AND (iParameterSet < 1 OR iParameterSet > 5) THEN		// invalid input for the parameter set
		xDownloadDone := FALSE; 
		xDownloadError := TRUE; 
		iResponse := eTransferResponse.invalid_ParameterSet; 
		iCurrentValue := 0; 
		// send command 'stop'
		fbWriteValueToWord(iValue := 61, iStartBit := 0, iEndBit := 5, wDataWord := awBusDataToVTEM[0]); 			// ValveMode = 61
		fbWriteValueToWord(iValue := 0, iStartBit := 6, iEndBit := 15, wDataWord := awBusDataToVTEM[0]); 			// (empty)
		awBusDataToVTEM[1] := 0; 
		awBusDataToVTEM[2] := 0; 
		
	ELSE	
		// call the function block for multiple parameter download
		fbdownloadMultipleParameters(	xExecute := xExecute,
										awBusDataFromVTEM := awBusDataFromVTEM,
										aTransferPackages := aTransferPackages, 
										awBusDataToVTEM := awBusDataToVTEM,
										xDownloadDone => xDownloadDone,
										xDownloadError => xDownloadError,
										iResponse => iResponse,
										iCurrentValue => iCurrentValue);
	END_IF
	
	
// The current value output is needed if there is any invalid value in order to address it correctly.
// As the user doesn't work with indices in this function block, the current value is transformed to a string holding the name of the parameter.
	CASE iCurrentValue OF
		0: sCurrentValue := 'iOperatingMode';
		1: sCurrentValue := 'iInPortRetract_optional';
		2: sCurrentValue := 'iInPortAdvanced_optional';
		3: sCurrentValue := 'AllParametersWritten';
	END_CASE

END_FUNCTION_BLOCK

